TYPE ST_UN_Machine100_Config :
STRUCT
	// Digital inputs
	// n.a.
	
	// Digital outputs
	// n.a.
	
	// Alarms
	// n.a.

	// Others
	// n.a.
	
END_STRUCT
END_TYPE

(* stored: Version 1.1.0.1, ProductVersion 3.1.4024.10
   DUT ST_UN_Machine100_Config: Id {d74f6583-f218-4d3f-b1ff-b01515744b9a} *)
